TYPE T_Ctrl_SIf_BCH_Par :
STRUCT
END_STRUCT
END_TYPE

(* stored: Version 1.1.0.1, ProductVersion 3.1.0.26
   DUT T_Ctrl_SIf_BCH_Par: Id {e3777b1d-a485-441e-8de6-ab9bdac44976} *)
